{attribute 'reflection'}
FUNCTION_BLOCK PUBLIC Fb_DevAxis EXTENDS FB_DevBase
VAR_INPUT
	// ===== General Function input =====
		fCmdAcc			: LREAL := 15000;
		fCmdDecc		: LREAL := 15000; 
	// ===== Master Axis =====
		refMasterAxis	: REFERENCE TO AXIS_REF ; // Master axis reference (if applicable)
		bReverseSlave	: BOOL 	:= FALSE; // Reverse slave axis relative to master
		fCmdGearRatio	: LREAL := 1 ; // Gear ratio Master/Slave (1/Ratio) 
	// Manual control reference
		stManualCtrl	: UDT_ManualAxisCtrl ;
END_VAR
VAR_OUTPUT
	// ====== State indications =======
		bHomed			: BOOL 	:= FALSE; 
		bError 			: BOOL 	:= FALSE;
		bStopped		: BOOL 	:= FALSE;
		bGearedAsSlave	: BOOL 	:= FALSE;
		bVelocityLimited: BOOL 	:= FALSE;  
		bIdle			: BOOL 	:= FALSE;
		fVelocity		: LREAL	:= 0	; // Axis velocity [rpm or units/sec] depending on config
		fActPosition	: LREAL := 0	; // Axis actual position [Units] depending on config	
		bReInTargetPos	: BOOL 	:= false; // rising edge axis is in position
	// ====== axis reference ======
		AxisRef			: AXIS_REF	; // Axis reference to hardware 
	// ====== Axis Settings ======
		fMaxVelo		: LREAL := 0 ; // Axis Maximum velocity
		fMaxAcc			: LREAL := 0 ; // Axis Maximum cceleration
		fMaxDec			: LREAL := 0 ; // axis Maxium deceleration 
	
		fSafeVeloLimit	: LREAL	:= 200; // Safe velocity limit 
		tEnableDelay	: TIME 	:= T#0MS	;
		tDisableDelay	: TIME 	:= T#500MS  ;
	// ==== Axis data ====
		fEncoderTurnoverValue	: LREAL ;   
END_VAR
VAR // Axis configuration 
	// ===== HW Config Bits =====
		bIcfCmdVelocityRpm	: BOOL ; // input speeds in Rpm
		bIcfEnableForward 	: BOOL ; // Enable forward motion
 		bIcfEnablereverse	: BOOL ; // Enable reverse motion
		bIcfAlwaysEnable	: BOOL ; // 1 = Axis always enabled, 0 = Axis disabled at Idle 
		bIcfSimulationMode	: BOOL := FALSE ; // Simulation mode is active [default set to False] 
		bIcfModuloAxis		: BOOL := FALSE ; // Show axis position as modulo
	// ===== Internal motion values ======
		fHomePosition		: LREAL := 0 ; // set position at homing
	// Command Modes
		mcHomingMode 		: MC_HomingMode := MC_direct ; // Homing Mode ( MC_DefaultHoming, MC_Direct, MC_ForceCallibration, MC_ResetCallibration)
	// Values from system
		McReadSysVelo		: MC_ReadParameter		; // Read Acceleration parameter from drive 
		McReadSysAcc		: MC_ReadParameter		; // Read Acceleration parameter from drive 
		McReadSysDec		: MC_ReadParameter		; // Read Acceleration parameter from drive 
END_VAR
VAR	// ====== Axis enable =====
		bCmdEnableAxis 		: BOOL 	:= FALSE; // Command to enable the axis (External)
		bInternalEnable		: BOOL 	:= FALSE; // internal enable command (turns off after set time, and on at new motion command
		bDelayedEnable		: BOOL 	:= false; // Delayed enable signal for motion commands
		TonMotionEnable		: TON 			; // Timer on for motion command enable
		TofIntAxisEnable	: TOF  			; // Timer off for internal axis enable 
	// Parameter read status 
		Cmd_EnDriveParRead	: BOOL 			; // Enable parameter read 
	// ===== Physical Homing signal =====
		IAxisHome AT %I* 	: BOOL 			; // Axis homing sensor from PLC (if MC_DefaultHoming is used)
END_VAR
VAR	// =============== Motion status functions ================
		fbMcReadAxisStatus	: MC_ReadStatus ;	// Fb for reading axis status	
	// =============== Motion function blocks =================
		fbMcPower 			: MC_Power		;		// FB for enable and override
		fbMcReset 			: MC_Reset		;		// FB to reset axis
		fbSoeReset			: FB_SoEReset	; 		// FB to reset axis hardware
		fbMcHome			: MC_Home		;		// Fb to home Axis
		fbMcStop 			: MC_Stop		;		// FB to stop axis
		fbMcHalt			: MC_Halt		;		// FB to halt axis
		fbMcJog				: MC_Jog		;		// FB to Jog axis
		fbMcMoveVelocity	: MC_MoveVelocity;		// FB to move with specified velocity until Next command is given
		fbMcGearInSlave		: MC_GearIn		;		// FB to gear axis to master 
		fbMcGearInDyn		: MC_GearInDyn	;		// FB to gear axis dynamicly to master
		fbMcGearOutSlave	: MC_GearOut	;		// FB to decouple gearing
		fbMcSetPosition		: MC_SetPosition;		// FB to Set axis position
//		fbMcWriteParameter	: MC_WriteParameterPersistent ; // FB to write parameters in persistend data

	(* PtoP Motion move commands are in arrays so multiple commands can be stacked *) 
		fbMCMoveRelative	: ARRAY [0..1] OF MC_MoveRelative	;		// FB to move relative
		fbMcMoveAbsolute	: ARRAY [0..1] OF MC_MoveAbsolute	;		// FB to move axis (velocity movement)
		fbMcMoveModulo		: ARRAY [0..1] OF MC_MoveModulo		;		// FB to move axis to modulo position
	// ===== Safe commands =====
		bCmdSafeStop	: BOOL ;
		bCmdSafeSpeed	: BOOL ; 
	// ===== Function execute triggers =====
		bExec_Reset			: BOOL := FALSE; // Execute reset
		bExec_Halt			: BOOL := FALSE; // Execute hold
		bExec_Home			: BOOL := FALSE; // Execute Home
		bExec_JogPositive	: BOOL := FALSE; // Execute Jog in positive direction
		bExec_JogNegative	: BOOL := FALSE; // Execute Jog in negative direction
		bExec_MoveVelocity	: BOOL := FALSE; // Execute move velocity
		bExec_GearAsSlave	: BOOL := FALSE; // Execute gear as slave
		bExec_GearSlaveDyn	: BOOL := FALSE; // Execute gear slave dynamic
		bExec_GearOutSlave	: BOOL := FALSE; // Execute gear out slave
		bExec_SetPosition	: BOOL := FALSE; // execute set position
//		bExec_ParWritePers	: BOOL := FALSE; // Execute parameter write persistent 
		
	// ===== Move ristrictions ======
		bCmdLimitVelocity 	: BOOL := FALSE			; // velocity limiting is active 
		fCmdVelocityLimit	: LREAL:= fSafeVeloLimit; // Maximum velocity limit when velocity limiting is active  
	(* PtoP Motion move commands are in arrays so multiple commands can be stacked *) 
		arExec_MoveRelative	: ARRAY [0..1] OF BOOL ; // Execute move relative
		arExec_MoveAbs		: ARRAY [0..1] OF BOOL ; // Execute move absolute reverse
		arExec_MoveModulo	: ARRAY [0..1] OF BOOL ; // Execute move modulo

	// ===== Internal variables =======
		fAcceleration	: LREAL := 0 ; // Acceleration used for functions 
		fDeceleration	: LREAL := 0 ; // Deceleration used for functions
END_VAR
VAR
	// ===== Loop variables =====
		i : DINT := 0 ; // For loop increment
	// ===== check variable ======
		rtrigInPosition	: R_TRIG ; // in position trigger
	// ===== Par write timer ===== 
END_VAR
VAR // Parameters 
	ParAccManualScaling	: Udt_Parameter := (fValue := 50, fFactory := 50, bTeachable := FALSE)  ; // Acceleration scaling factor for manual functions 
	ParDecManualScaling	: Udt_Parameter := (fValue := 50, fFactory := 50, bTeachable := FALSE)	; // Deceleration scaling factor for manual functions 
END_VAR

// Call base function
SUPER^(refFbFault := refFbFault);

// ==== Check if axis is initiated =====
IF NOT bInitOk THEN 
	RETURN ; 
END_IF

// ===== Execute safe functions =====
	ExecSafeFunctions(); 
	
// ==== Execute organizational functions =====
	CallOrganizationFunctions();

// ==== execute motion functions =====
	CallMotionFunctions();

METHOD PRIVATE CallMotionFunctions : BOOL
VAR_INPUT
END_VAR
// ===== Check if safe to move =====
	IF (bManual AND bSafetyOk) THEN
		;
	ELSIF bCmdSafeStop THEN 
		// ===== reset safe commands ======
		bCmdSafeStop	:= FALSE ; 
		RETURN ;
	END_IF

// ===== Set acceleratio and deceleration values =======
	IF bCmdManual THEN 
		fAcceleration 	:= fCmdAcc * (ParAccManualScaling.fvalue / 100);
		fDeceleration	:= fCmdDecc* (ParDecManualScaling.fValue / 100);
	END_IF
// ===== Homing functions =====
	ExecHome		(); 

// ===== Motion standstil commands =====
	ExecHalt		();

// ===== Motion move functions
	ExecJog			(); 
	ExecMoveAbsolute();
	ExecMoveRelative();
	ExecMoveModulo	();
	ExecMoveVelocity();
	
// ===== Execute gearing functions =====
	ExecGearOut		();
	ExecGearIn		();
	ExecGearDynamic	();
	
// ====== reset velocity lmiting =====
	bVelocityLimited	:= bCmdLimitVelocity ;	
	bCmdLimitVelocity 	:= FALSE ; 

// ====== Reset acceleration deceleration values ======
	fAcceleration	:= fCmdAcc;
	fDeceleration	:= fCmdDecc;
END_METHOD

METHOD PRIVATE CallOrganizationFunctions : BOOL
VAR_INPUT
END_VAR
// ==== execute organizational functions =====
	ExecReadStatus		(); 
	ExecEnable			();
	ExecReset			();
//	ExecWriteParameter	();
	ExecSetPosition		();
END_METHOD

METHOD PUBLIC CmdGearDynamic : BOOL // Set axis to geared, activates with variable gear ratio until geared out or stopped (if method is no longer called then gear ratio is locked to last value)
VAR_INPUT
	fGearRatio	:	LREAL	:= 1	; // Slave Axis gearing ratio (Master = 1/ fGearRatio = Slave)	
END_VAR
// set blocked command if halt is active 
bBlockedCommand := fbMcHalt.Active ;

// Set command to true 
bExec_GearSlaveDyn 	:= TRUE ;
bInternalEnable		:= TRUE ;

// coppy parameters
fCmdGearRatio 				:= fGearRatio ;

// Set feedback output 
CmdGearDynamic := fbMcGearInDyn.Active ;
END_METHOD

METHOD PUBLIC CmdGearIn : BOOL // Set axis to geared, activates with constant gear ratio until geared out or stopped
VAR_INPUT
	fGearRatio	:	LREAL	:= 1	; // Slave Axis gearing ratio (Master = 1/ fGearRatio = Slave)	
END_VAR
// set blocked command if halt is active 
bBlockedCommand := fbMcHalt.Active ;

// Set command to true 
bExec_GearAsSlave 	:= TRUE ;
bInternalEnable		:= TRUE ;

// coppy parameters
fCmdGearRatio 				:= fGearRatio ;

// Set feedback output 
CmdGearIn := fbMcGearInSlave.Active ;
END_METHOD

METHOD CmdGearOut : BOOL
VAR_INPUT
END_VAR
// set blocked command if halt is active 
bBlockedCommand := fbMcHalt.Active ;

// Set command to true
bExec_GearOutSlave 	:= TRUE ;
bExec_GearAsSlave	:= FALSE;
bExec_GearSlaveDyn 	:= FALSE;

// Set feedback Output
CmdGearOut := fbMcGearOutSlave.Done;
END_METHOD

METHOD PUBLIC CmdHalt : BOOL
VAR_INPUT
	fDeceleration 	: LREAL := 0 ; // command deceleration
	mcBuffermode	: MC_BufferMode ; // Buffermode defines how the previous command is executed.
END_VAR
// Set command to true 
bExec_Halt 		:= TRUE ;
bInternalEnable	:= TRUE ;

// coppy parameters
fbMcHalt.Deceleration	:= fDeceleration;
fbMcHalt.BufferMode		:= mcBuffermode	;

// Set feedback output 
CmdHalt := fbMchalt.Active OR fbMcHalt.Done ;
END_METHOD

METHOD PUBLIC CmdHome : BOOL // start axis homing procedure
VAR_INPUT
	fPosition 		: LREAL := 0 ; // Homing position
END_VAR
// set blocked command if halt is active 
bBlockedCommand := fbMcHalt.Active ;

// set command to true 
bExec_Home 		:= TRUE	; 
bInternalEnable	:= TRUE ;

// coppy parameters
fbMcHome.Position 	:= fPosition 	;

// Set feedback output
CmdHome := fbMcHome.Done ;
END_METHOD

METHOD PUBLIC CmdJog : BOOL // Jog axis with variable speed. jog stops as soon as the command is false
VAR_INPUT
	fVelocity		: LREAL 	; // jog velocity can be adjusted as long as the command is active
	fPos			: LREAL 	; // Jog position or step size (if aplicable)
	bJogNegative 	: BOOL 		:= FALSE ; // jog in negative direction
	eJogmode		: E_JogMode := E_JogMode.MC_JOGMODE_CONTINOUS ; // jogmode [default MC_JOGMODE_CONTINOUS] 
END_VAR
// set blocked command if halt is active 
bBlockedCommand := fbMcHalt.Active ;

// Velocity conversion from RPM to deg/sec
	IF bIcfCmdVelocityRpm THEN 
		fVelocity := Rpm_To_DegS(fVelocity);
	END_IF

// Set command to true
	IF fbMcJog.Velocity = fVelocity THEN // If command velocity changes, then set exec to false for one cycle to trigger new velocity so the jog follows the set velocity
		bExec_JogPositive	:= NOT bJogNegative ;
		bExec_JogNegative 	:= bJogNegative ;
	END_IF
	bInternalEnable			:= TRUE ;

// coppy parameters
	fbMcJog.Velocity	:= fVelocity 	;
	fbmcjog.Mode		:= eJogmode		;
	fbMcJog.Position	:= fPos			;

// Set feedback output 
	CmdJog := fbMcJog.Active ;
END_METHOD

METHOD PUBLIC CmdLimitVelocity : BOOL // limit axis maximum velocity, stays active as long as command is called. 
VAR_INPUT
	fVelocityLimit	: LREAL ; // velocity Maximum limit
END_VAR
// set blocked command if halt is active 
bBlockedCommand := fbMcHalt.Active ;

// Set velocity limiting command 
bCmdLimitVelocity S= TRUE;
	
// Set velocity maximum value 
fCmdVelocityLimit := fVelocityLimit ; 

// set feedback 
CmdLimitVelocity := bVelocityLimited ;
END_METHOD

METHOD PUBLIC CmdManual : BOOL
VAR
	eJogmode		: E_JogMode := E_JogMode.MC_JOGMODE_CONTINOUS ; // jogging mode 
END_VAR
// set blocked command if halt is active 
bBlockedCommand := fbMcHalt.Active ;

// Enable axis for manual control
bCmdManual := TRUE ;

// check safety 
IF NOT bSafetyOk THEN 
	RETURN;
END_IF

// set jog mode 
IF stManualCtrl.bCmdInching THEN 
	eJogmode := E_JogMode.MC_JOGMODE_INCHING ;
END_IF

// execute motion commands
IF stManualCtrl.bCmdJogForward OR stManualCtrl.bCmdJogReverse THEN 
	CmdJog (fVelocity := stManualCtrl.fVelocity, 
			fPos := stManualCtrl.fDistance, 
			bJogNegative := stManualCtrl.bCmdJogReverse, 
			eJogmode := eJogmode);
ELSIF stManualCtrl.bCmdToPos THEN 
	CmdMoveAbs( fPosition := stManualCtrl.fPosition, 
				fVelocity := stManualCtrl.fVelocity, 
				mcBuffermode := MC_BufferMode.MC_Aborting);
ELSIF stManualCtrl.bCmdHome THEN 
	CmdHome( fPosition := 0);
ELSE 
	CmdHalt( 	fDeceleration := fMaxDec * 0.9, 
				mcBuffermode := MC_BufferMode.MC_Aborting) ; 
END_IF
END_METHOD

METHOD PUBLIC CmdMoveAbs : BOOL // Move absolute command
VAR_INPUT
	fPosition	:	LREAL 	; // target position
	fVelocity	: 	LREAL 	; // Maximum velocity [units/sec]
	mcBuffermode: 	MC_BufferMode ; // Buffermode defines how the previous command is executed.
END_VAR
// set blocked command if halt is active 
bBlockedCommand := fbMcHalt.Active ;

// Velocity conversion from RPM to deg/sec
	IF bIcfCmdVelocityRpm THEN 
		fVelocity := Rpm_To_DegS(fVelocity);
	END_IF

// Determine function for command stacking
	IF fbMcMoveAbsolute[0].Active THEN 
		arExec_MoveAbs[1] 				:= (fPosition <> fbMcMoveAbsolute[0].Position OR fVelocity <> fbMcMoveAbsolute[0].Velocity) ;
		fbMcMoveAbsolute[1].Position 	:= fPosition ;
		fbMcMoveAbsolute[1].Velocity 	:= fVelocity ; 
		fbMcMoveAbsolute[1].BufferMode 	:= mcBuffermode ;
	ELSE
		arExec_MoveAbs[0] 				:= (fPosition <> fbMcMoveAbsolute[1].Position OR fVelocity <> fbMcMoveAbsolute[1].Velocity) ;
		fbMcMoveAbsolute[0].Position 	:= fPosition ;
		fbMcMoveAbsolute[0].Velocity 	:= fVelocity ; 
		fbMcMoveAbsolute[0].BufferMode 	:= mcBuffermode ;
	END_IF

bInternalEnable	:= TRUE ;

// set feedback
IF arExec_MoveAbs[1] OR fbMcMoveAbsolute[1].Busy THEN 
	CmdMoveAbs :=	fbMcMoveAbsolute[1].Active ;
ELSE 
	CmdMoveAbs :=	fbMcMoveAbsolute[0].Active ;
END_IF
END_METHOD

METHOD PUBLIC CmdMoveModulo : BOOL // Move to a modulo position
VAR_INPUT
	fPosition	:	LREAL 	; // target position
	fVelocity	: 	LREAL 	; // Maximum velocity [units/sec]
	mcDirection : 	MC_Direction := MC_Direction.MC_Positive_Direction ; // Direction of movement mc_direction [ deafult mc_positive_direction]
	mcBuffermode: 	MC_BufferMode ; // Buffermode defines how the previous command is executed.
END_VAR
// set blocked command if halt is active 
bBlockedCommand := fbMcHalt.Active ;

// Velocity conversion from RPM to deg/sec
	IF bIcfCmdVelocityRpm THEN 
		fVelocity := Rpm_To_DegS(fVelocity);
	END_IF

// Determine function for command stacking
	IF fbMcMoveModulo[0].Active THEN 
		arExec_MoveModulo[1] 		:= (fPosition <> fbMcMoveModulo[0].Position OR fVelocity <> fbMcMoveModulo[0].Velocity)	;
		fbMcMoveModulo[1].Velocity 	:= fVelocity 	;
		fbMcMoveModulo[1].Position 	:= fPosition 	;
		fbMcMoveModulo[1].Direction	:= mcDirection	;
		fbMcMoveModulo[1].BufferMode:= mcBuffermode ;
	ELSE    
		arExec_MoveModulo[0] 		:= (fPosition <> fbMcMoveModulo[1].Position OR fVelocity <> fbMcMoveModulo[1].Velocity) ;
		fbMcMoveModulo[0].Velocity 	:= fVelocity 	;
		fbMcMoveModulo[0].Position 	:= fPosition 	;
		fbMcMoveModulo[0].Direction	:= mcDirection	;
		fbMcMoveModulo[0].BufferMode:= mcBuffermode ;
	END_IF

bInternalEnable	:= TRUE ;

(*// Reset position position and velocity commands
	IF fbMcMoveModulo[1].Active AND NOT fbMcMoveModulo[0].Busy THEN 
		fbMcMoveModulo[0].Velocity := 0 ;
		fbMcMoveModulo[0].Position := 0 ;
	ELSIF fbMcMoveModulo[0].Active AND NOT fbMcMoveModulo[1].Busy THEN 
		fbMcMoveModulo[1].Velocity := 0 ;
		fbMcMoveModulo[1].Position := 0 ;
 	END_IF 
*)
// set feedback
IF arExec_MoveModulo[1] OR fbMcMoveModulo[1].Busy THEN 
	CmdMoveModulo :=	fbMcMoveModulo[1].Active OR fbMcMoveModulo[1].Done;
ELSE
	CmdMoveModulo :=	fbMcMoveModulo[0].Active OR fbMcMoveModulo[0].Done ;
END_IF
END_METHOD

METHOD CmdMoveRelative : BOOL // move relative command 
VAR_INPUT
	fDistance	:	LREAL 	; // target position
	fVelocity	: 	LREAL 	; // Maximum velocity [units/sec]
	mcBuffermode: 	MC_BufferMode ; // Buffermode defines how the previous command is executed.
END_VAR
// set blocked command if halt is active 
bBlockedCommand := fbMcHalt.Active ;

// Velocity conversion from RPM to deg/sec
	IF bIcfCmdVelocityRpm THEN 
		fVelocity := Rpm_To_DegS(fVelocity);
	END_IF

// Determine function for command stacking
	IF fbMCMoveRelative[0].Active THEN 
		arExec_MoveRelative[1] := (fDistance <> fbMCMoveRelative[0].Distance OR fVelocity <> fbMCMoveRelative[0].Velocity) ;
		fbMCMoveRelative[1].Velocity	:= fVelocity 	;
		fbMCMoveRelative[1].Distance	:= fDistance	;
		fbMCMoveRelative[1].BufferMode	:= mcBuffermode	;
	ELSE 
		arExec_MoveRelative[0] := (fDistance <> fbMCMoveRelative[1].Distance OR fVelocity <> fbMCMoveRelative[1].Velocity) ;
		fbMCMoveRelative[0].Velocity	:= fVelocity 	;
		fbMCMoveRelative[0].Distance	:= fDistance	;
		fbMCMoveRelative[0].BufferMode	:= mcBuffermode	;
	END_IF

bInternalEnable	:= TRUE ;

// set feedback
IF arExec_MoveRelative[1] OR fbMCMoveRelative[1].Busy THEN 
	CmdMoveRelative :=	fbMCMoveRelative[1].Active ;
ELSE
	CmdMoveRelative :=	fbMCMoveRelative[0].Active ;
END_IF
END_METHOD

METHOD PUBLIC CmdMoveVelocity : BOOL // Move with set velocity until stopped
VAR_INPUT
	fVelocity	: 	LREAL 	; // Maximum velocity [units/sec]
	mcDirection : 	MC_Direction := MC_Direction.MC_Positive_Direction ; // Direction of movement mc_direction [ deafult mc_positive_direction]
	mcBuffermode: 	MC_BufferMode ; // Buffermode defines how the previous command is executed.
END_VAR
// set blocked command if halt is active 
bBlockedCommand := fbMcHalt.Active ;

// Velocity conversion from RPM to deg/sec
	IF bIcfCmdVelocityRpm THEN 
		fVelocity := Rpm_To_DegS(fVelocity);
	END_IF

// Set command to true 
	bExec_MoveVelocity 	:= TRUE ;
	bInternalEnable		:= TRUE ;

// coppy parameters
	fbMcMoveVelocity.Velocity	:= fVelocity 	;
	fbMcMoveVelocity.Direction 	:= mcDirection	;
	fbMcMoveVelocity.BufferMode	:= mcBuffermode	;

// Set feedback output 
	CmdMoveVelocity := fbMcMoveVelocity.Active ;
END_METHOD

METHOD PUBLIC CmdOverwriteAcc : BOOL // temporarilly overwrite deceleration values
VAR_INPUT	
	fValue	: LREAL ; // Overwrite value 
END_VAR
fAcceleration := fValue ;

CmdOverwriteAcc := TRUE ;
END_METHOD

METHOD PUBLIC CmdOverwriteDec : BOOL // Temporarilly overwrite deceleration values
VAR_INPUT
	fValue	: LREAL ; // Overwrite value 
END_VAR
fDeceleration := fValue ;

CmdOverwriteDec := TRUE ;
END_METHOD

METHOD PUBLIC CmdReset : BOOL
VAR_INPUT
END_VAR
// set blocked command if halt is active 
bBlockedCommand := fbMcHalt.Active ;

// Set reset axis to true 				
	bExec_Reset 	:= TRUE ; 
	bInternalEnable	:= TRUE ;
	
// Set feedback output 
	CmdReset := fbMcReset.Done ;
END_METHOD

METHOD PUBLIC CmdSafeSpeed : BOOL
VAR_INPUT
END_VAR
// Set safestop command
bCmdSafeSpeed := TRUE ; 

// Set feedback output 
CmdSafeSpeed := AxisRef.NcToPlc.ActVelo <= fSafeVeloLimit ;
END_METHOD

METHOD PUBLIC CmdSafeStop : BOOL
VAR_INPUT
END_VAR

// Set safestop command
bCmdSafeStop := TRUE ; 

// Set feedback output 
CmdSafeStop := bIsSafe OR NOT bInitOk;
END_METHOD

METHOD PUBLIC CmdSetPosition : BOOL
VAR_INPUT
	fPosition		: LREAL ; // encoder position
	bSetRelative	: BOOL 	; // TRUE = relative position offset, FALSE = Absolute position
END_VAR
bExec_SetPosition 			:= NOT fbMcSetPosition.Busy AND NOT fbMcSetPosition.Done ; 
fbMcSetPosition.Position	:= fPosition ;
fbMcSetPosition.Mode		:= bSetRelative ;

CmdSetPosition := fbMcSetPosition.Done;
END_METHOD

METHOD PRIVATE ExecEnable : BOOL
VAR_INPUT
END_VAR
// ===== Set axis enable ======
IF bCmdManual AND bSafetyOk THEN 
	bCmdEnableAxis 	:= TRUE ;
	bInternalEnable S= bCmdManual ;
	bCmdManual 		:= FALSE ;
ELSIF NOT bEnable AND AxisRef.Status.Moving THEN
	CmdHalt(fDeceleration := fCmdDecc, mcBuffermode := MC_BufferMode.MC_Aborting);
ELSE 
	bCmdEnableAxis	:= bEnable  ;
END_IF

// ===== Check if axis is bussy with a command =====
	bInternalEnable S= AxisRef.Status.HasJob;
	bInternalEnable	S= bIcfAlwaysEnable ; // always enable axis if configured
	bInternalEnable	S= AxisRef.Status.Coupled ;
	
// ===== Axis disable timer after last command =====
	TofIntAxisEnable (	IN:= bInternalEnable, PT := tDisableDelay);

// ===== check if parameter write is not busy =====
//	bCmdEnableAxis R= bExec_ParWritePers OR fbMcWriteParameter.Busy;
	
// ===== Enable drive =====
	fbMcPower(	Axis			:= AxisRef , 
				Enable			:= bCmdEnableAxis AND TofIntAxisEnable.Q, 
				Enable_Positive	:= bIcfEnableForward, 
				Enable_Negative	:= bIcfEnablereverse, 
				Override		:= 100 );  
				
// ===== Reset internal enable signal =====
	bInternalEnable := FALSE ; 	

// ===== Delayed enable function =====	
	TonMotionEnable(IN := fbMcPower.Status, PT := tEnableDelay);
	bDelayedEnable := TonMotionEnable.Q ;	


IF fbMcPower.Error THEN 
	bError					:= TRUE							;
	stFault.Active 			:= TRUE 						;
	stFault.MessageNumber	:= E_MessageNumbers.FF_AxisFault;
	stFault.Discription		:= CONCAT('Enable Fault ', UDINT_TO_STRING(fbMcPower.ErrorID));
	stFault.Discription		:= CONCAT( sName , stfault.Discription ) ;
	stFault.FaultType		:= E_FaultTypes.FF				;
END_IF
END_METHOD

METHOD INTERNAL ExecGearDynamic : BOOL
VAR_INPUT
END_VAR
// ===== invert gear ratio if reverse slave is active =====
	IF bReverseSlave THEN 
		fbMcGearInDyn.GearRatio := fCmdGearRatio * -1 ;
	ELSE 
		fbMcGearInDyn.GearRatio := fCmdGearRatio ;
	END_IF

// ===== Execute gear in function =====
	fbMcGearInDyn ( 	Master 			:= refMasterAxis,
						Slave			:= AxisRef,
						Enable 			:= bExec_GearSlaveDyn AND bDelayedEnable,
						Acceleration	:= fAcceleration	); 
						
// ===== reset command =====
	bExec_GearSlaveDyn	:= FALSE ;
	bGearedAsSlave		:= fbMcGearInDyn.InGear ; 

// Gearing fault handling 
	IF fbMcGearInDyn.Error THEN 
		bError					:= TRUE							;
		stFault.Active 			:= TRUE 						;
		stFault.MessageNumber	:= E_MessageNumbers.FF_AxisFault;
		stFault.Discription		:= CONCAT('Gear dynamic Fault ', UDINT_TO_STRING(fbMcGearInDyn.ErrorID));	
		stFault.Discription		:= CONCAT( sName , stfault.Discription ) ;
		stFault.FaultType		:= E_FaultTypes.FF				;
	END_IF
END_METHOD

METHOD INTERNAL ExecGearIn : BOOL
VAR_INPUT
END_VAR
// ===== invert gear ratio if reverse slave is active =====
	IF bReverseSlave THEN 
		fbMcGearInSlave.RatioNumerator := fCmdGearRatio * -1 ;
	ELSE 
		fbMcGearInSlave.RatioNumerator := fCmdGearRatio ;
	END_IF

// ===== Execute gear in function =====
	fbMcGearInSlave ( 	Master 			:= refMasterAxis,
						Slave			:= AxisRef,
						Execute 		:= bExec_GearAsSlave AND bDelayedEnable,
						RatioDenominator:= 1	); 
						
// ===== reset command =====
	bExec_GearAsSlave 	:= FALSE  ;
	bGearedAsSlave		S= fbMcGearInSlave.InGear ; 

// Gearing fault handling 
	IF fbMcGearInSlave.Error THEN 
		bError					:= TRUE							;
		stFault.Active 			:= TRUE 						;
		stFault.MessageNumber	:= E_MessageNumbers.FF_AxisFault;
		stFault.Discription		:= CONCAT('Gear as slave Fault ', UDINT_TO_STRING(fbMcGearInSlave.ErrorID));
		stFault.Discription		:= CONCAT( sName , stfault.Discription ) ;
		stFault.FaultType		:= E_FaultTypes.FF				;
	END_IF
END_METHOD

METHOD INTERNAL ExecGearOut : BOOL
VAR_INPUT
END_VAR
// ===== execute gear out function ======
	fbMcGearOutSlave (	Slave 	:= AxisRef,
						Execute := bExec_GearOutSlave );

// ===== reset command =====
	bExec_GearOutSlave	:= false ;
	bGearedAsSlave		R= fbMcGearOutSlave.Done 	; 

// Gearing fault handling 
	IF fbMcGearOutSlave.Error THEN 
		bError					:= TRUE							;
		stFault.Active 			:= TRUE 						;
		stFault.MessageNumber	:= E_MessageNumbers.FF_AxisFault;
		stFault.Discription		:= CONCAT('Gear out Fault ', UDINT_TO_STRING(fbMcGearOutSlave.ErrorID));
		stFault.Discription		:= CONCAT( sName , stfault.Discription ) ;
		stFault.FaultType		:= E_FaultTypes.FF				;
	END_IF
END_METHOD

METHOD INTERNAL ExecHalt : BOOL
VAR_INPUT
END_VAR
// ==== Execute halt function ===== 
fbMcHalt (	Axis 		:= AxisRef,
			Execute 	:= bExec_Halt );

// ===== reset command =====
	bExec_Halt := FALSE ;
	
// Halt fault handling 
	IF fbMcHalt.Error THEN 
		bError					:= TRUE							;
		stFault.Active 			:= TRUE 						;
		stFault.MessageNumber	:= E_MessageNumbers.FF_AxisFault;
		stFault.Discription		:= CONCAT('Halt Fault ', UDINT_TO_STRING(fbMcHalt.ErrorID));
		stFault.Discription		:= CONCAT( sName , stfault.Discription ) ;
		stFault.FaultType		:= E_FaultTypes.FF				;
	END_IF
END_METHOD

METHOD INTERNAL ExecHome : BOOL
VAR_INPUT
END_VAR
// ==== execute homing function =====
	fbMcHome(	Axis			:= AxisRef,
				Execute			:= bExec_Home AND bDelayedEnable,
				HomingMode		:= mcHomingMode,
				bCalibrationCam	:= IAxisHome ); 
			
// Reset exec command 
	bExec_Home 	:= FALSE ;
	bHomed		S= fbMcHome.Done ;	
				
// fault handling 
	IF fbMcHome.Error THEN 
		bError					:= TRUE							;
		stFault.Active 			:= TRUE 						;
		stFault.MessageNumber	:= E_MessageNumbers.FF_AxisFault;
		stFault.Discription		:= CONCAT('Homing Fault ', UDINT_TO_STRING(fbMcHome.ErrorID));
		stFault.Discription		:= CONCAT( sName , stfault.Discription ) ;
		stFault.FaultType		:= E_FaultTypes.FF				;
	END_IF
END_METHOD

METHOD INTERNAL ExecJog : BOOL
VAR_INPUT
END_VAR
// ===== Execute Jog function =====
	// velocity limiting
		IF bCmdSafeSpeed THEN 
			fbMcJog.Velocity := MIN(fSafeVeloLimit, fbMcJog.Velocity); 
		ELSIF bCmdLimitVelocity THEN 
			fbMcJog.Velocity := MIN(fCmdVelocityLimit, fbMcJog.Velocity); 
		END_IF
	// function call
	fbMcJog (	Axis 		:= AxisRef,
				JogForward	:= bExec_JogPositive AND bDelayedEnable,
				JogBackwards:= bExec_JogNegative AND bDelayedEnable,
				Acceleration:= fAcceleration,
				Deceleration:= fDeceleration );

// ===== reset command =====
	bExec_JogPositive 	:= FALSE  ;
	bExec_JogNegative	:= FALSE  ;
	
// Jog fault handling 
	IF fbMcJog.Error THEN 
		bError					:= TRUE							;
		stFault.Active 			:= TRUE 						;
		stFault.MessageNumber	:= E_MessageNumbers.FF_AxisFault;
		stFault.Discription		:= CONCAT('Jog Fault ', UDINT_TO_STRING(fbMcJog.ErrorID));
		stFault.Discription		:= CONCAT( sName , stfault.Discription ) ;
		stFault.FaultType		:= E_FaultTypes.FF				;
	END_IF
END_METHOD

METHOD INTERNAL ExecMoveAbsolute : BOOL
VAR_INPUT
END_VAR
// ==== execute move absolute function =====
FOR i := 0 TO 1 DO 
	// velocity limiting
		IF bCmdSafeSpeed THEN 
			fbMcMoveAbsolute[i].Velocity := MIN(fSafeVeloLimit, fbMcMoveAbsolute[i].Velocity); 
		ELSIF bCmdLimitVelocity THEN 
			fbMcMoveAbsolute[i].Velocity := MIN(fCmdVelocityLimit, fbMcMoveAbsolute[i].Velocity); 
		END_IF
	// function call
	fbMcMoveAbsolute[i](	Axis 		:= AxisRef,
							Execute 	:= arExec_MoveAbs[i] AND bDelayedEnable,
							Acceleration:= fAcceleration,
							Deceleration:= fDeceleration );  

	// If function is done then reset command values
	IF fbMcMoveAbsolute[i].Done OR fbMcMoveAbsolute[i].CommandAborted OR NOT arExec_MoveAbs[i] THEN 
		fbMcMoveAbsolute[i].Velocity	:= 0 ;
		fbMcMoveAbsolute[i].Position	:= 0 ; 
	END_IF

	// reset Exec command 
	arExec_MoveAbs[i] := FALSE ; 
	
	// fault handling 
	IF fbMcMoveAbsolute[i].Error THEN 
		bError					:= TRUE							;
		stFault.Active 			:= TRUE 						;
		stFault.MessageNumber	:= E_MessageNumbers.FF_AxisFault;
		stFault.Discription		:= CONCAT('Move absolute Fault ', UDINT_TO_STRING(fbMcMoveAbsolute[i].ErrorID));
		stFault.Discription		:= CONCAT( sName , stfault.Discription ) ;
		stFault.FaultType		:= E_FaultTypes.FF				;
	END_IF
END_FOR
END_METHOD

METHOD INTERNAL ExecMoveModulo : BOOL
VAR_INPUT
END_VAR
// ===== Execute move modulo function =====
FOR i := 0 TO 1 DO 
	// velocity limiting
		IF bCmdSafeSpeed THEN 
			fbMcMoveModulo[i].Velocity := MIN(fSafeVeloLimit, fbMcMoveModulo[i].Velocity); 
		ELSIF bCmdLimitVelocity THEN 
			fbMcMoveModulo[i].Velocity := MIN(fCmdVelocityLimit, fbMcMoveModulo[i].Velocity); 
		END_IF
	// function call
	fbMcMoveModulo[i](	Axis 		:= AxisRef,
						Execute 	:= arExec_MoveModulo[i] AND bDelayedEnable,
						Acceleration:= fAcceleration,
						Deceleration:= fDeceleration);  
	
	// If function is done then reset command values
	IF fbMcMoveModulo[i].Done OR fbMcMoveModulo[i].CommandAborted OR NOT arExec_MoveModulo[i] THEN 
		fbMcMoveModulo[i].Velocity	:= 0 ;
		fbMcMoveModulo[i].Position	:= 0 ; 
	END_IF

	// reset Exec command 
	arExec_MoveModulo[i] := FALSE ; 
	
	// fault handling 
	IF fbMcMoveModulo[i].Error THEN 
		bError					:= TRUE							;
		stFault.Active 			:= TRUE 						;
		stFault.MessageNumber	:= E_MessageNumbers.FF_AxisFault;
		stFault.Discription		:= CONCAT('Move module Fault ', UDINT_TO_STRING(fbMcMoveModulo[i].ErrorID));
		stFault.Discription		:= CONCAT( sName , stfault.Discription ) ;
		stFault.FaultType		:= E_FaultTypes.FF			;
	END_IF
END_FOR
END_METHOD

METHOD INTERNAL ExecMoveRelative : BOOL
VAR_INPUT
END_VAR
// ===== Execute move relative function ======
FOR i := 0 TO 1 DO 
	// velocity limiting
		IF bCmdSafeSpeed THEN 
			fbMCMoveRelative[i].Velocity := MIN(fSafeVeloLimit, fbMCMoveRelative[i].Velocity); 
		ELSIF bCmdLimitVelocity THEN 
			fbMCMoveRelative[i].Velocity := MIN(fCmdVelocityLimit, fbMCMoveRelative[i].Velocity); 
		END_IF
	// function call
	fbMCMoveRelative[i](	Axis 		:= AxisRef,
							Execute		:= arExec_MoveRelative[i] AND bDelayedEnable,
							Acceleration:= fAcceleration,
							Deceleration:= fDeceleration );

	// If function is done then reset command values
	IF fbMCMoveRelative[i].Done OR fbMCMoveRelative[i].CommandAborted OR NOT arExec_MoveRelative[i] THEN 
		fbMCMoveRelative[i].Velocity	:= 0 ;
		fbMCMoveRelative[i].Distance	:= 0 ; 
	END_IF

	// reset Exec command 
	arExec_MoveRelative[i] := FALSE ; 
	
	// fault handling 
	IF fbMCMoveRelative[i].Error THEN 
		bError					:= TRUE							;
		stFault.Active 			:= TRUE 						;
		stFault.MessageNumber	:= E_MessageNumbers.FF_AxisFault;
		stFault.Discription		:= CONCAT('Move relative Fault ', UDINT_TO_STRING(fbMCMoveRelative[i].ErrorID));
		stFault.Discription		:= CONCAT( sName , stfault.Discription ) ;
		stFault.FaultType		:= E_FaultTypes.FF			;
	END_IF
END_FOR
END_METHOD

METHOD INTERNAL ExecMoveVelocity : BOOL
VAR_INPUT
END_VAR
// ===== Execute move velocity function =====
// velocity limiting
IF bCmdSafeSpeed THEN 
	fbMcMoveVelocity.Velocity := MIN(fSafeVeloLimit, fbMcMoveVelocity.Velocity); 
ELSIF bCmdLimitVelocity THEN 
	fbMcMoveVelocity.Velocity := MIN(fCmdVelocityLimit, fbMcMoveVelocity.Velocity); 
END_IF
// function call
fbMcMoveVelocity (	Axis 		:= AxisRef,
					Execute		:= bExec_MoveVelocity  AND bDelayedEnable,
					Acceleration:= fAcceleration,
					Deceleration:= fDeceleration );

// ===== reset command =====
bExec_MoveVelocity := FALSE ;
	
// Halt fault handling 
IF fbMcMoveVelocity.Error THEN 
	bError					:= TRUE							;
	stFault.Active 			:= TRUE 						;
	stFault.MessageNumber	:= E_MessageNumbers.FF_AxisFault;
	stFault.Discription		:= CONCAT('Move velocity Fault ', UDINT_TO_STRING(fbMcMoveVelocity.ErrorID));
	stFault.Discription		:= CONCAT( sName , stfault.Discription ) ;
	stFault.FaultType		:= E_FaultTypes.FF				;
END_IF
END_METHOD

METHOD INTERNAL ExecReadStatus : BOOL
VAR_INPUT
END_VAR
// Read axis status from drive
fbMcReadAxisStatus (	Enable 	:= TRUE ,
						Axis 	:= AxisRef );
						
// convert velocity to RPM for output if aplicable
IF bIcfCmdVelocityRpm THEN 
	fVelocity := AxisRef.NcToPlc.ActVelo / 6 ;
ELSE 
	fVelocity := AxisRef.NcToPlc.ActVelo ;
END_IF

// write position output
IF bIcfModuloAxis THEN 
	fActPosition := AxisRef.NcToPlc.ModuloActPos ;
ELSE
	fActPosition := AxisRef.NcToPlc.ActPos ;
END_IF
						
// set status bits 
bIdle := NOT AxisRef.Status.HasJob ;

// read fault handling 
IF fbMcReadAxisStatus.Error THEN 
	bError					:= TRUE							;
	stFault.Active 			:= TRUE 						;
	stFault.MessageNumber	:= E_MessageNumbers.FF_AxisFault;
	stFault.Discription		:= CONCAT('Status read fault ', UDINT_TO_STRING(fbMcPower.ErrorID));
	stFault.Discription		:= CONCAT( sName , stfault.Discription ) ;
	stFault.FaultType		:= E_FaultTypes.FF				;
END_IF

// In position 
	rtrigInPosition( 	CLK := AxisRef.Status.InTargetPosition, 
						Q => bReInTargetPos);
END_METHOD

METHOD INTERNAL ExecReset : BOOL
VAR_INPUT
END_VAR
IF  AxisRef.Status.Moving AND bExec_Reset THEN // If the axis is still moving execute safe stop first
	CmdSafeStop();
	RETURN;
END_IF

// ===== Reset axis, drive and axis functions =====
	fbSoeReset ( 	Execute := bExec_Reset AND NOT fbMcReset.Busy AND NOT bIcfSimulationMode, // No physical drive reset necesarry when not connected 
					Timeout := T#10S		,
					Axis	:= AxisRef		);
	
	fbMcReset	( 	Execute	:= bexec_reset AND NOT fbSoeReset.Busy,
					Axis	:= AxisRef ); 
					
// ===== reset command =====
	bExec_Reset := FALSE ;
	
// ===== reset internal fault bits and stop bits =====
	bError 			:= FALSE ; 
	
// Reset fault handling 
	IF fbSoeReset.Error OR fbMcReset.Error THEN 
		bError					:= TRUE							;
		stFault.Active 			:= TRUE 						;
		stFault.MessageNumber	:= E_MessageNumbers.FF_AxisFault;
		stFault.Discription		:= CONCAT('Reset Fault ', UDINT_TO_STRING(fbMcReset.ErrorID));
		stFault.Discription		:= CONCAT( sName , stfault.Discription ) ;
		stFault.FaultType		:= E_FaultTypes.FF				;
	END_IF
END_METHOD

METHOD PRIVATE ExecSafeFunctions : BOOL
VAR_INPUT
END_VAR
// ==== Stop when safety is not ok =====
	bCmdSafeStop S= NOT bSafetyOk ;

// ==== Safe operation functions (overrule all other motion functions) =====
	fbMcStop( 	Axis 			:= AxisRef		,
				Execute 		:= bCmdSafeStop	,
				Deceleration	:= fMaxDec		);
	
	// Reset axis command			
	bCmdSafeStop 	R= fbMcStop.Done OR AxisRef.Status.HasBeenStopped ;
	bStopped		:= AxisRef.Status.HasBeenStopped ;

// Safestop fault handling 
	IF fbMcStop.Error THEN 
		bError					:= TRUE							;
		stFault.Active 			:= TRUE 						;
		stFault.MessageNumber	:= E_MessageNumbers.FF_AxisFault;
		stFault.Discription		:= CONCAT('Safe stop axis fault ', UDINT_TO_STRING(fbMcStop.ErrorID));
		stFault.Discription		:= CONCAT( sName , stfault.Discription ) ;
		stFault.FaultType		:= E_FaultTypes.FF				;
	END_IF
	
// ===== Safe speed monitoring =====
	IF bCmdSafeSpeed THEN 
		IF AxisRef.NcToPlc.ActVelo > fSafeVeloLimit THEN 
			bExec_Halt := TRUE ; 
			ExecHalt(); 
		ELSE 
			bCmdSafeSpeed := FALSE ; 
		END_IF
	END_IF

// ===== Dev is safe feedback =====
bIsSafe := AxisRef.Status.HasBeenStopped  ;
END_METHOD

METHOD INTERNAL ExecSetPosition : BOOL
VAR_INPUT
END_VAR
// ====== set position of axis ======
IF bExec_SetPosition OR fbMcSetPosition.Busy THEN 
	fbMcSetPosition (	Axis 	:= AxisRef,
						Execute	:= bExec_SetPosition );
	bExec_SetPosition := TRUE ;
END_IF
END_METHOD

METHOD PRIVATE ExecWriteParameter : BOOL
VAR_INPUT
END_VAR
// check if axis is disabled before writeing parameter
	AxisRef.ReadStatus();
	IF AxisRef.Status.Disabled 
	AND (fbMcWriteParameter.Busy OR bExec_ParWritePers) THEN
		fbMcWriteParameter	( 	Axis 	:= AxisRef,
								Execute	:= bExec_ParWritePers );
	ELSE
		fbMcWriteParameter.Execute := FALSE ; 
		RETURN;
	END_IF
						
// fault handling 
	IF fbMcWriteParameter.Error THEN 
		bError					:= TRUE							;
		stFault.Active 			:= TRUE 						;
		stFault.MessageNumber	:= E_MessageNumbers.FF_AxisFault;
		stFault.Discription		:= CONCAT('Cannot write parameter Id#:', UDINT_TO_STRING(fbMcHome.ErrorID));
		stFault.Discription		:= CONCAT( sName , stfault.Discription ) ;
		stFault.FaultType		:= E_FaultTypes.FF				;
	END_IF
 
// reset commands
	bExec_ParWritePers := FALSE ;
END_METHOD

METHOD PUBLIC Init : BOOL
VAR_INPUT
	// Message location data
	nId			: UDINT ; // Identification number of object
	nParentId	: UDINT ; // Id of higher level If aplicable (0 = no parent)
	// Config Bits
	bIcfCmdVelocityRpm	: BOOL := FALSE ; // input speeds in Rpm
	bIcfEnableForward 	: BOOL := TRUE 	; // Enable forward motion
	bIcfEnablereverse	: BOOL := TRUE 	; // Enable reverse motion
	bIcfAlwaysEnable	: BOOL := FALSE ; // 1 = Axis always enabled, 0 = Axis disabled at Idle 
	bIcfSimulationMode	: BOOL := FALSE ; // Simulation mode is active [default set to False] Used for testing without hardware present 
	bIcfModuloAxis		: BOOL := FALSE ; // Show axis position as modulo
	
	// Config Values 
	mcHomingMode 		: MC_HomingMode := MC_HomingMode.MC_DefaultHoming; 
	fHomePosition		: LREAL := 0 	; // set position at homing
	fSafeVeloLimit		: LREAL	:= 360 	; // safe velocity limit [deg/sec]
	nEncTurnoverVal 	: LREAL := 360	; // encoder turnover value 
	tEnableDelay		: time 	:= T#0MS; // Time between axis enable command and motion command execution (0 := no delay active)	
	tDisabledelay		: TIME 	:= T#100MS; // Axis idle time before axis is disabled 
END_VAR
VAR 
	bActVeloReadValid 	: BOOL ; // velocity parameter read is valid 
	bActAccReadValid 	: BOOL ; // Acceleration parameter read is valid 
	bActDecReadValid 	: BOOL ; // Deceleration parameter read is valid 
	bActParamValid 		: BOOL ; // Parameter read is valid 
END_VAR
// ====== Calculate device id =====
	ExecIdentifyDevice(nId,nParentId, E_ComponentTypes.Axis);

// ====== Set manual device type ======
	eDevType := E_Devices.Axis ;	
	
// ===== Message data set =====
	stFault.ComponentType		:= E_ComponentTypes.Axis ;
	
// ===== Read system configuration =====
	McReadSysVelo	(	Axis 			:= AxisRef,
						Enable 			:= Cmd_EnDriveParRead ,
						ParameterNumber := MaxVelocitySystem ,
						ReadMode		:= 1,
						Valid			=> bActVeloReadValid ,						
						Busy			=> ,
						Error			=> ,
						ErrorID			=> ,
						Value			=> fMaxVelo );
	McReadSysAcc	(	Axis 			:= AxisRef,
						Enable 			:= Cmd_EnDriveParRead ,
						ParameterNumber := MaxAccelerationSystem ,
						ReadMode		:= 1,
						Valid			=> bActAccReadValid ,						
						Busy			=> ,
						Error			=> ,
						ErrorID			=> ,
						Value			=> fMaxAcc );
	McReadSysDec	(	Axis 			:= AxisRef,
						Enable 			:= Cmd_EnDriveParRead ,
						ParameterNumber := MaxDecelerationSystem ,
						ReadMode		:= 1,
						Valid			=> bActDecReadValid ,						
						Busy			=> ,
						Error			=> ,
						ErrorID			=> ,
						Value			=> fMaxDec );

	IF 	fMaxVelo > 0 
	AND fMaxAcc >0
	AND fMaxDec >0 THEN 
		bActParamValid	:= TRUE ; 
		fCmdAcc 		:= fMaxAcc * 0.9;
		fCmdDecc		:= fMaxDec * 0.9;
	END_IF

	IF NOT Cmd_EnDriveParRead AND NOT bActParamValid THEN  
		Cmd_EnDriveParRead := TRUE;
	ELSIF Cmd_EnDriveParRead THEN
		Cmd_EnDriveParRead := FALSE;
	END_IF

// ===== Configure Axis =====
	// ***** Config Bits *****
		THIS^.bIcfCmdVelocityRpm	:= bIcfCmdVelocityRpm	; // Enable speed inputs in Rpm
		THIS^.bIcfEnableForward 	:= bIcfEnableForward 	; // Enable forward motion
		THIS^.bIcfEnablereverse		:= bIcfEnablereverse	; // Enable reverse motion
		THIS^.bIcfAlwaysEnable		:= bIcfAlwaysEnable		; // Always enable motor and brake if safety is ok
		THIS^.bIcfSimulationMode	:= bIcfSimulationMode 	; // Simulation mode is active [default set to False] 
		THIS^.bIcfModuloAxis		:= bIcfModuloAxis		; // show axis position as modulo

	// ***** config homing Mode ***** 
 		THIS^.mcHomingMode 			:= mcHomingMode ; // set homing mode
		THIS^.fHomePosition			:= fHomePosition;
	// ***** Velocity settings *****
		THIS^.fSafeVeloLimit 		:= fSafeVeloLimit ; // set maximum safe velocity	
	// ***** Encoder values *****
		THIS^.fEncoderTurnoverValue := nEncTurnoverVal	; // turnover value for encoder = 25.6 mm per rev * 4096 revolutions 
	// ***** Time delay enable off *****
		THIS^.tEnableDelay		:= tEnableDelay	;
		THIS^.tDisableDelay 	:= tDisabledelay ;		
		
// ===== configure parameters =====
	ParAccManualScaling.fMinimum 		:= 1 	;
	ParAccManualScaling.fMaximum		:= 100 	;
	ParAccManualScaling.nNumber 		:= nLocationId + 1;
	ParAccManualScaling.sDiscription  	:= CONCAT( STR1 := sName, STR2 := 'percantage of acceleration used For jogging');
	ParAccManualScaling.sName			:= CONCAT( STR1 := sName, STR2 := 'Manual acc scaling');
	ParAccManualScaling.sType			:= 'Mpar';
	ParAccManualScaling.sUnit			:= '%';

	ParDecManualScaling.fMinimum 		:= 1 	;
	ParDecManualScaling.fMaximum		:= 100 	;
	ParDecManualScaling.nNumber 		:= nLocationId + 2;
	ParDecManualScaling.sDiscription  	:= CONCAT( STR1 := sName, STR2 := 'percantage of deceleration used For jogging');
	ParDecManualScaling.sName			:= CONCAT( STR1 := sName, STR2 := 'Manual dec scaling');
	ParDecManualScaling.sType			:= 'Mpar';
	ParDecManualScaling.sUnit			:= '%';
		
// ===== reset axis state indicators ======
	bError 	:= FALSE;

// ====== Set init to done =======
IF bActParamValid THEN 
	bInitOk	:= TRUE ; 
END_IF
END_METHOD

END_FUNCTION_BLOCK

(* stored: Version 1.1.0.1, ProductVersion 3.1.4024.5
   POU Fb_DevAxis: Id {bc69e9b9-3f3d-4df5-a0a1-a0954c261e17}, SpecialFunc None
   Folder Command Methods: Id {e50539d8-81cc-4181-8633-d48ea6a3afe6}
   Folder Private: Id {5a5a8788-fda6-4189-8936-e923757baeb9}
   Folder Motion: Id {8c2ebe7c-f13d-4e72-aa37-ecee84af7d2f}
   Folder Organization: Id {b45159df-0aaf-4b82-b633-88517773f7ca}
   Method CallMotionFunctions: Id {e3f4db07-f896-41c6-b4ce-2c24a2a65ee1}
   Method CallOrganizationFunctions: Id {30788d1f-d292-49da-a183-d882588243a9}
   Method CmdGearDynamic: Id {7011281c-220c-4832-81a9-6de31a7ec1a3}
   Method CmdGearIn: Id {d39d912d-cd60-47f9-9c58-f4c673b83377}
   Method CmdGearOut: Id {0eba1dc5-045c-4e71-9b15-315cb2debe34}
   Method CmdHalt: Id {76ed2c19-987b-01bf-2d8e-dfce06b9fc82}
   Method CmdHome: Id {9156a5be-9684-4b33-891a-938949533f96}
   Method CmdJog: Id {19a0b1de-6384-40c6-bca2-fc0bfb1b6d9a}
   Method CmdLimitVelocity: Id {5d066d54-5fea-4b4f-abf4-5d71884c951d}
   Method CmdManual: Id {bc280ce4-7b96-06c9-0aff-4a50ef532241}
   Method CmdMoveAbs: Id {897ddefe-6fd9-4aa0-8e52-b781b66bb019}
   Method CmdMoveModulo: Id {8d63fd5b-c612-4ee0-92e7-3eb778fa38f1}
   Method CmdMoveRelative: Id {2ed540a9-f0c6-4ad5-b603-5e75ef38aff1}
   Method CmdMoveVelocity: Id {87d516ce-706c-45c2-bb7f-438c77a1a8af}
   Method CmdOverwriteAcc: Id {0bcd5b3c-1fc1-0254-21e2-286bd45e95c0}
   Method CmdOverwriteDec: Id {d18160bd-16ee-085d-3a89-64c41286e618}
   Method CmdReset: Id {9ed88b7b-6fd1-4ff9-a6de-53b6c8907919}
   Method CmdSafeSpeed: Id {ddc13036-fa7e-46f4-be16-22a24c1d346b}
   Method CmdSafeStop: Id {b3ad69e2-24fe-00d4-08f1-72f39343c002}
   Method CmdSetPosition: Id {cdd58728-eb33-090b-146a-18a5bc82ad75}
   Method ExecEnable: Id {97d17d4c-4218-4969-bb76-cf3660f2ac5b}
   Method ExecGearDynamic: Id {a5fd620e-146f-471b-9689-dc40fdcad502}
   Method ExecGearIn: Id {0347e51e-7471-437a-a77d-dd0ede1aed70}
   Method ExecGearOut: Id {137dca5b-ff36-41d7-8d1e-db831854f7be}
   Method ExecHalt: Id {b37253d8-5f2a-4031-b9a5-f7589796c62b}
   Method ExecHome: Id {e9c8969e-9f26-46cc-b798-0ff95ca0c652}
   Method ExecJog: Id {f7873e37-f6a3-45f7-a57d-76a2b3d914bd}
   Method ExecMoveAbsolute: Id {c32ad101-c406-42f7-900a-821300c800d0}
   Method ExecMoveModulo: Id {ddd8d330-0e54-4a84-b928-b81d871d62c3}
   Method ExecMoveRelative: Id {ff02329f-50f4-404d-ae21-618dca212cb3}
   Method ExecMoveVelocity: Id {d07f3661-ff1b-448e-89ce-6edde810b751}
   Method ExecReadStatus: Id {bcfefbac-5e3a-4829-b533-395a75a11713}
   Method ExecReset: Id {289eb010-9ce0-40f7-84c2-391c18144f9a}
   Method ExecSafeFunctions: Id {de6e8394-dce8-4579-9944-987f245a933f}
   Method ExecSetPosition: Id {42f95ac0-57d0-06e7-037d-d914ca0d57d6}
   Method ExecWriteParameter: Id {e25e6df9-2845-09eb-3e44-2acd7fb0470d}
   Method Init: Id {0a8c2089-518e-4a9f-9c10-83a2f8fbff86} *)
